(* IEC 61131-3 sources: eCockpitGit/test_project/src/%F%00 Library/%F%Common Functions/%F%MinMax, 10 files *)

(* ---- %POU%FU_bMinMaxValue.st ---- *)
//This function keeps a variable between a minimum and a maximum value
// +-----------+----------+----------+-----------------------------------------------------------------------------------------------------------------------+
// |**Version**|**Author**| **Date** |**Changes**                                                                                                            |
// +-----------+----------+----------+-----------------------------------------------------------------------------------------------------------------------+
// | 1         | NSN      | 07-01-18 | Creation                                                                                                              |
// +-----------+----------+----------+-----------------------------------------------------------------------------------------------------------------------+
FUNCTION FU_bMinMaxValue : BOOL
VAR_IN_OUT
	Variable		:BYTE;
END_VAR
VAR_INPUT
	MinVal			:BYTE;
	MaxVal			:BYTE;
END_VAR
(*%!%__DELIMITER__%!%*)
IF Variable < MinVal THEN			//This makes sure only values between 0 and 10000 can be entered
	Variable				:=		MinVal;
ELSIF Variable > MaxVal THEN
	Variable				:=		MaxVal;
END_IF

(* ---- %POU%FU_diMinMaxValue.st ---- *)
//This function keeps a variable between a minimum and a maximum value
// +-----------+----------+----------+-----------------------------------------------------------------------------------------------------------------------+
// |**Version**|**Author**| **Date** |**Changes**                                                                                                            |
// +-----------+----------+----------+-----------------------------------------------------------------------------------------------------------------------+
// | 1         | NSN      | 07-01-18 | Creation                                                                                                              |
// +-----------+----------+----------+-----------------------------------------------------------------------------------------------------------------------+
FUNCTION FU_diMinMaxValue : BOOL
VAR_IN_OUT
	Variable		:DINT;
END_VAR
VAR_INPUT
	MinVal			:DINT;
	MaxVal			:DINT;
END_VAR
(*%!%__DELIMITER__%!%*)
IF Variable < MinVal THEN			//This makes sure only values between 0 and 10000 can be entered
	Variable				:=		MinVal;
ELSIF Variable > MaxVal THEN
	Variable				:=		MaxVal;
END_IF

(* ---- %POU%FU_dwMinMaxValue.st ---- *)
//This function keeps a variable between a minimum and a maximum value
// +-----------+----------+----------+-----------------------------------------------------------------------------------------------------------------------+
// |**Version**|**Author**| **Date** |**Changes**                                                                                                            |
// +-----------+----------+----------+-----------------------------------------------------------------------------------------------------------------------+
// | 1         | NSN      | 07-01-18 | Creation                                                                                                              |
// +-----------+----------+----------+-----------------------------------------------------------------------------------------------------------------------+
FUNCTION FU_dwMinMaxValue : BOOL
VAR_IN_OUT
	Variable		:DWORD;
END_VAR
VAR_INPUT
	MinVal			:DWORD;
	MaxVal			:DWORD;
END_VAR
(*%!%__DELIMITER__%!%*)
IF Variable < MinVal THEN			//This makes sure only values between 0 and 10000 can be entered
	Variable				:=		MinVal;
ELSIF Variable > MaxVal THEN
	Variable				:=		MaxVal;
END_IF

(* ---- %POU%FU_iMinMaxValue.st ---- *)
//This function keeps a variable between a minimum and a maximum value
// +-----------+----------+----------+-----------------------------------------------------------------------------------------------------------------------+
// |**Version**|**Author**| **Date** |**Changes**                                                                                                            |
// +-----------+----------+----------+-----------------------------------------------------------------------------------------------------------------------+
// | 1         | NSN      | 07-01-18 | Creation                                                                                                              |
// +-----------+----------+----------+-----------------------------------------------------------------------------------------------------------------------+
FUNCTION FU_iMinMaxValue : BOOL
VAR_IN_OUT
	Variable		:INT;
END_VAR
VAR_INPUT
	MinVal			:INT;
	MaxVal			:INT;
END_VAR
(*%!%__DELIMITER__%!%*)
IF Variable < MinVal THEN			//This makes sure only values between 0 and 10000 can be entered
	Variable				:=		MinVal;
ELSIF Variable > MaxVal THEN
	Variable				:=		MaxVal;
END_IF

(* ---- %POU%FU_rMinMaxValue.st ---- *)
//This function keeps a variable between a minimum and a maximum value
// +-----------+----------+----------+-----------------------------------------------------------------------------------------------------------------------+
// |**Version**|**Author**| **Date** |**Changes**                                                                                                            |
// +-----------+----------+----------+-----------------------------------------------------------------------------------------------------------------------+
// | 1         | NSN      | 07-01-18 | Creation                                                                                                              |
// +-----------+----------+----------+-----------------------------------------------------------------------------------------------------------------------+
FUNCTION FU_rMinMaxValue : BOOL
VAR_IN_OUT
	Variable		:REAL;
END_VAR
VAR_INPUT
	MinVal			:REAL;
	MaxVal			:REAL;
END_VAR
(*%!%__DELIMITER__%!%*)
IF Variable < MinVal THEN			//This makes sure only values between minval and maxval can be entered
	Variable				:=		MinVal;
ELSIF Variable > MaxVal THEN
	Variable				:=		MaxVal;
END_IF

(* ---- %POU%FU_siMinMaxValue.st ---- *)
//This function keeps a variable between a minimum and a maximum value
// +-----------+----------+----------+-----------------------------------------------------------------------------------------------------------------------+
// |**Version**|**Author**| **Date** |**Changes**                                                                                                            |
// +-----------+----------+----------+-----------------------------------------------------------------------------------------------------------------------+
// | 1         | NSN      | 07-01-18 | Creation                                                                                                              |
// +-----------+----------+----------+-----------------------------------------------------------------------------------------------------------------------+
FUNCTION FU_siMinMaxValue : BOOL
VAR_IN_OUT
	Variable		:SINT;
END_VAR
VAR_INPUT
	MinVal			:SINT;
	MaxVal			:SINT;
END_VAR
(*%!%__DELIMITER__%!%*)
IF Variable < MinVal THEN			//This makes sure only values between 0 and 10000 can be entered
	Variable				:=		MinVal;
ELSIF Variable > MaxVal THEN
	Variable				:=		MaxVal;
END_IF

(* ---- %POU%FU_udiMinMaxValue.st ---- *)
//This function keeps a variable between a minimum and a maximum value
// +-----------+----------+----------+-----------------------------------------------------------------------------------------------------------------------+
// |**Version**|**Author**| **Date** |**Changes**                                                                                                            |
// +-----------+----------+----------+-----------------------------------------------------------------------------------------------------------------------+
// | 1         | NSN      | 07-01-18 | Creation                                                                                                              |
// +-----------+----------+----------+-----------------------------------------------------------------------------------------------------------------------+
FUNCTION FU_udiMinMaxValue : BOOL
VAR_IN_OUT
	Variable		:UDINT;
END_VAR
VAR_INPUT
	MinVal			:UDINT;
	MaxVal			:UDINT;
END_VAR
(*%!%__DELIMITER__%!%*)
IF Variable < MinVal THEN			//This makes sure only values between 0 and 10000 can be entered
	Variable				:=		MinVal;
ELSIF Variable > MaxVal THEN
	Variable				:=		MaxVal;
END_IF

(* ---- %POU%FU_uiMinMaxValue.st ---- *)
//This function keeps a variable between a minimum and a maximum value
// +-----------+----------+----------+-----------------------------------------------------------------------------------------------------------------------+
// |**Version**|**Author**| **Date** |**Changes**                                                                                                            |
// +-----------+----------+----------+-----------------------------------------------------------------------------------------------------------------------+
// | 1         | NSN      | 07-01-18 | Creation                                                                                                              |
// +-----------+----------+----------+-----------------------------------------------------------------------------------------------------------------------+
FUNCTION FU_uiMinMaxValue : BOOL
VAR_IN_OUT
	Variable		:UINT;
END_VAR
VAR_INPUT
	MinVal			:UINT;
	MaxVal			:UINT;
END_VAR
(*%!%__DELIMITER__%!%*)
IF Variable < MinVal THEN			//This makes sure only values between 0 and 10000 can be entered
	Variable				:=		MinVal;
ELSIF Variable > MaxVal THEN
	Variable				:=		MaxVal;
END_IF

(* ---- %POU%FU_usiMinMaxValue.st ---- *)
//This function keeps a variable between a minimum and a maximum value
// +-----------+----------+----------+-----------------------------------------------------------------------------------------------------------------------+
// |**Version**|**Author**| **Date** |**Changes**                                                                                                            |
// +-----------+----------+----------+-----------------------------------------------------------------------------------------------------------------------+
// | 1         | NSN      | 07-01-18 | Creation                                                                                                              |
// +-----------+----------+----------+-----------------------------------------------------------------------------------------------------------------------+
FUNCTION FU_usiMinMaxValue : BOOL
VAR_IN_OUT
	Variable		:USINT;
END_VAR
VAR_INPUT
	MinVal			:USINT;
	MaxVal			:USINT;
END_VAR
(*%!%__DELIMITER__%!%*)
IF Variable < MinVal THEN			//This makes sure only values between 0 and 10000 can be entered
	Variable				:=		MinVal;
ELSIF Variable > MaxVal THEN
	Variable				:=		MaxVal;
END_IF

(* ---- %POU%FU_wMinMaxValue.st ---- *)
//This function keeps a variable between a minimum and a maximum value
// +-----------+----------+----------+-----------------------------------------------------------------------------------------------------------------------+
// |**Version**|**Author**| **Date** |**Changes**                                                                                                            |
// +-----------+----------+----------+-----------------------------------------------------------------------------------------------------------------------+
// | 1         | NSN      | 07-01-18 | Creation                                                                                                              |
// +-----------+----------+----------+-----------------------------------------------------------------------------------------------------------------------+
FUNCTION FU_wMinMaxValue : BOOL
VAR_IN_OUT
	Variable		:WORD;
END_VAR
VAR_INPUT
	MinVal			:WORD;
	MaxVal			:WORD;
END_VAR
(*%!%__DELIMITER__%!%*)
IF Variable < MinVal THEN			//This makes sure only values between 0 and 10000 can be entered
	Variable				:=		MinVal;
ELSIF Variable > MaxVal THEN
	Variable				:=		MaxVal;
END_IF
